(* CoDeSys 2.3.9.59 project: C2_Struct_Array_To_CSV.pro *)
(* Libraries: Standard.lib, Util.lib 20.3.15 10:30:08, SysLibCallback.lib, SysLibSockets.lib, SysLibTasks.lib, SysLibRtc.lib, SysLibFile.lib, SysLibPlcCtrl.lib *)

(* Task configuration *)
TASK tskCsvFile (PRIORITY := 10, INTERVAL := T#100ms);
	PRG_EV2_Logger();
END_TASK
TASK tskMain (PRIORITY := 1, INTERVAL := T#20ms);
	PRG_MAIN();
END_TASK

(* Global variable list: Global_Variables *)
VAR_GLOBAL
	EtatVide : Struct_Etat_EV2 := (
		Etat_EV2_ON		:= FALSE,
		Etat_EV2_OFF	:= FALSE,
		DateTime_EV2	:= DT#1970-01-01-00:00:00
	);
END_VAR

(* Data type *)
TYPE Struct_Etat_EV2 :
STRUCT
	Etat_EV2_ON		: BOOL;
	Etat_EV2_OFF	: BOOL;
	DateTime_EV2	: DT;
END_STRUCT
END_TYPE

(* POU 10_PROG/PRG_EV2_Logger, ST *)
PROGRAM PRG_EV2_Logger
VAR
    i : INT;

    TrigON  : R_TRIG;
    TrigOFF : F_TRIG;

	TabEtat_EV2		: ARRAY[0..100] OF Struct_Etat_EV2;
	IndexTab_EV2	: INT := 0;

    Serializer : FB_EV2_Serializer;

    FileName : STRING(80);
    FileNum  : DWORD;
    Header   : STRING(80);

    SortieEV2 : BOOL; (* connecter à la vraie sortie *)
END_VAR
(* === Déclencheurs === *)
TrigON(CLK := SortieEV2);
TrigOFF(CLK := SortieEV2);

(* === Enregistrement tableau === *)
IF TrigON.Q THEN
    TabEtat_EV2[IndexTab_EV2].Etat_EV2_ON  := TRUE;
    TabEtat_EV2[IndexTab_EV2].Etat_EV2_OFF := FALSE;
    TabEtat_EV2[IndexTab_EV2].DateTime_EV2 := SysRtcGetTime(TRUE);
    IndexTab_EV2 := IndexTab_EV2 + 1;
END_IF;

IF TrigOFF.Q THEN
    TabEtat_EV2[IndexTab_EV2].Etat_EV2_ON  := FALSE;
    TabEtat_EV2[IndexTab_EV2].Etat_EV2_OFF := TRUE;
    TabEtat_EV2[IndexTab_EV2].DateTime_EV2 := SysRtcGetTime(TRUE);
    IndexTab_EV2 := IndexTab_EV2 + 1;
END_IF;

(* === Tableau plein === *)
IF IndexTab_EV2 > 100 THEN

    (* 1. Générer nom fichier *)
	FileName := '\InternalStorage\';				(* Inclusion du chemin *)
    FileName := CONCAT(FileName, BuildFileName());	(* Génération du nom de fichier horodaté *)

    (* 2. Ouvrir fichier *)
    FileNum := SysFileOpen(FileName, 'w');

    (* 3. Écrire header *)
    Header := 'EtatON;EtatOFF;DateTime$0D$0A';
    SysFileWrite(FileNum, ADR(Header), LEN(Header));

    (* 4. Écrire chaque ligne CSV *)
    FOR i := 0 TO 100 DO
        Serializer(Data := TabEtat_EV2[i]);
        SysFileWrite(FileNum, ADR(Serializer.CSVLine), LEN(Serializer.CSVLine));
    END_FOR;

    (* 5. Fermer le fichier *)
    SysFileClose(FileNum);

    (* 6. Réinitialiser tableau *)
    IndexTab_EV2 := 0;
    FOR i := 0 TO 100 DO
        TabEtat_EV2[i] := EtatVide;
    END_FOR;
END_IF;
END_PROGRAM

(* POU 30_FUNCTION BLOCK/FB_EV2_Serializer, ST *)
FUNCTION_BLOCK FB_EV2_Serializer
VAR_INPUT
    Data : Struct_Etat_EV2;
END_VAR

VAR_OUTPUT
    CSVLine : STRING(255);
END_VAR

VAR
    tmp : STRING(50);
END_VAR
CSVLine := '';

tmp := BOOL_TO_STRING(Data.Etat_EV2_ON);
CSVLine := CONCAT(CSVLine, tmp);
CSVLine := CONCAT(CSVLine, ';');

tmp := BOOL_TO_STRING(Data.Etat_EV2_OFF);
CSVLine := CONCAT(CSVLine, tmp);
CSVLine := CONCAT(CSVLine, ';');

tmp := DT_TO_STRING(Data.DateTime_EV2);
CSVLine := CONCAT(CSVLine, tmp);
CSVLine := CONCAT(CSVLine, '$0D$0A');
END_FUNCTION_BLOCK

(* POU 20_FUNCTION/BuildFileName, ST *)
FUNCTION BuildFileName : STRING(80)
VAR
    dtNow      : DT;
    dtString   : STRING(25);

    yearStr    : STRING(4);
    monthStr   : STRING(2);
    dayStr     : STRING(2);
    hourStr    : STRING(2);
    minStr     : STRING(2);
    secStr     : STRING(2);

    fileName   : STRING(80);
END_VAR
(* 1. Récupération DT actuel *)
dtNow := SysRtcGetTime(TRUE);

(* 2. Conversion DT -> STRING *)
dtString := DT_TO_STRING(dtNow);
(* Exemple : 'DT#2026-03-24-10:45:22' *)

(* 3. Extraction des sous-chaînes *)
yearStr  := MID(dtString, 4, 4);
monthStr := MID(dtString, 2, 9);
dayStr   := MID(dtString, 2, 12);
hourStr  := MID(dtString, 2, 15);
minStr   := MID(dtString, 2, 18);
secStr   := MID(dtString, 2, 21);

(* 4. Construction du nom de fichier *)
fileName := 'EV2_';
fileName := CONCAT(fileName, yearStr);
fileName := CONCAT(fileName, monthStr);
fileName := CONCAT(fileName, dayStr);
fileName := CONCAT(fileName, '_');
fileName := CONCAT(fileName, hourStr);
fileName := CONCAT(fileName, minStr);
fileName := CONCAT(fileName, secStr);
fileName := CONCAT(fileName, '.csv');

BuildFileName := fileName;
END_FUNCTION

(* POU 10_PROG/PRG_MAIN, ST *)
PROGRAM PRG_MAIN
VAR
END_VAR
;
END_PROGRAM

(* POU 00_README/README, ST *)
PROGRAM README
VAR
END_VAR
(* === README =====================================================================================

PROCESS
"""""""

1. Remplissage du tableau au fil des événements

	À chaque changement d’état EV2 :

	- On remplit *une ligne* du tableau "TabEtat_EV2[Index]"
	- On incrémente "Index"

2. Lorsque "Index" = 100 on bascule en creation de fichier .csv

	- On génère le nom de fichier incluant le chemin et un horadatage pour éviter d'écraser le précédent
	- On ouvre le nouveau fichier
	- On écrit l'entête (optionnel)
	- On entre dans une boucle qui écrit cahque ligne l'une après l'autre
	- On referme le fichier
	- On réinitialise le tableau "TabEtat_EV2[Index]"

NOTA
""""

Le chemin (path) dépend de la destination du fichier .csv

	- \InternalStorage\
	- \StorageCard\
	- \UsbStorage\

================================================================================================ *)
;
END_PROGRAM
